FUNCTION_BLOCK FB_SITP_SygnalizacjaStanu IMPLEMENTS ITF_SITP_SygnalizacjaStanu
VAR
	refarrLampki				: REFERENCE TO ARRAY [1..STALE.ILOSC_LAMPEK_SYGNALIZACYJNYCH] OF B_IO.ITF_LampkaRozszerzona;
END_VAR

METHOD PUBLIC PowiazTablice
VAR_INPUT
	refarrLampki				: REFERENCE TO ARRAY [1..STALE.ILOSC_LAMPEK_SYGNALIZACYJNYCH] OF B_IO.ITF_LampkaRozszerzona;
END_VAR
THIS^.refarrLampki				REF= refarrLampki;
END_METHOD

METHOD PUBLIC UstawPrace
VAR_INPUT

END_VAR
END_METHOD

METHOD PUBLIC Wylacz
VAR_INPUT
	eLampka				: E_SITP_LampkiSygnalizacyjne;
END_VAR
THIS^.refarrLampki [eLampka].Wylacz ();
END_METHOD

METHOD PUBLIC WylaczWszystkie
VAR_INPUT
END_VAR

VAR
	iI: INT;
END_VAR
FOR iI := 1 TO STALE.ILOSC_LAMPEK_SYGNALIZACYJNYCH DO
	THIS^.refarrLampki [iI].Wylacz ();
END_FOR
END_METHOD

METHOD PUBLIC ZwrocStan : BOOL
VAR_INPUT
	eLampka			 : E_SITP_LampkiSygnalizacyjne;
END_VAR
ZwrocStan			:= THIS^.refarrLampki [eLampka].Stan ();
END_METHOD

END_FUNCTION_BLOCK

(* stored: Version 1.1.0.1
   POU FB_SITP_SygnalizacjaStanu: Id {cbc3efe0-f491-0759-1bd6-b19e42623d30}, SpecialFunc None
   Method PowiazTablice: Id {d114f5b5-e3b6-008d-2491-c02d11ce7efa}
   Method UstawPrace: Id {064623cb-3cfc-039b-2598-74bd5eb004e9}
   Method Wylacz: Id {c6c6e1c8-86ad-0ed0-0291-63ccb6115850}
   Method WylaczWszystkie: Id {51a5cf19-9ea1-0b0d-2b20-67a02c3d7852}
   Method ZwrocStan: Id {f1565313-e360-0045-2428-720cb83cced2} *)
